KUKA KRL program: Up23.src, Up23.dat

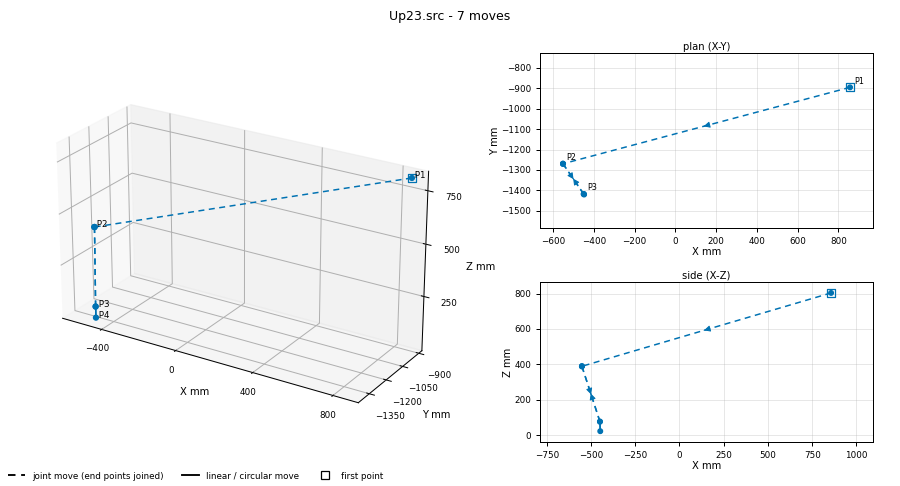
[picture p0: tool path of Up23.src, 7 of 7 moves have a stored position in this frame; points joined in program order, loops and branches not executed]
--- Up23.src ---
&ACCESS RV1
&REL 151
&COMMENT VW380 Ablegen_AFO415600
&PARAM EDITMASK = Up999[1-999]
&PARAM TPVW_VERSION = 8.3.18
&PARAM TEMPLATE = C:\KRC\Roboter\Template\upvorgabe
&PARAM DISKPATH = UPs
DEF UP23()
   ; FOLD UP Anfang;%{SE} %MKUKATPVW
   SPS_N=-1
   SPS_FERTIG=FALSE
   IF NOT CALLBYSELECT THEN
      INTERRUPT DECL 10 WHEN $CYCFLAG[254]==FALSE DO VW(#FB_STOP,TRUE)
      INTERRUPT ON 10
      INT10=TRUE
      VW_USR_R (#USR_INIT)
   ENDIF
   VW(#VW_INIT_UP,TRUE)
   ; ENDFOLD
   ;FOLD -- VW380, THIL -- ;%{PSE}%MKUKATPVW,%CVW_COM,%VCOMMENT,%P 1:Comment:, 2:VW380, THIL
      ;FOLD {H}
         M_COMMENT("VW380, THIL")
      ;ENDFOLD
   ;ENDFOLD
   ;FOLD -- 415600R01 -- ;%{PSE}%MKUKATPVW,%CVW_COM,%VCOMMENT,%P 1:Comment:, 2:415600R01
      ;FOLD {H}
         M_COMMENT("415600R01")
      ;ENDFOLD
   ;ENDFOLD
   ;FOLD -- FRG ST415600 -- ;%{PSE}%MKUKATPVW,%CVW_COM,%VCOMMENT,%P 1:Comment:, 2:FRG ST415600
      ;FOLD {H}
         M_COMMENT("FRG ST415600")
      ;ENDFOLD
   ;ENDFOLD
   ;FOLD -- ACHTUNG! Position ist nicht von PF0 anfahrbar! -- ;%{PSE}%MKUKATPVW,%CVW_COM,%VCOMMENT,%P 1:Comment:, 2:ACHTUNG! Position ist nicht von PF0 anfahrbar!
      ;FOLD {H}
         M_COMMENT("ACHTUNG! Position ist nicht von PF0 anfahrbar!")
      ;ENDFOLD
   ;ENDFOLD
   ;FOLD PTP VB=100% VE=0% ACC=100% RobWzg=11 Base=0 SPSTrig=0[1/100s] P ;%{P}%MKUKATPVW,%CMOVE8,%VPTP,%P 1:1, 2: VB=, 3:100, 4:%, 5: VE=, 6:0, 7:%, 8: ACC=, 9:100, 10:%, 11: RobWzg=, 12:11, 13: Base=, 14:0, 15: SPSTrig=, 16:0, 17:[1/100s], 18: P, 19:1, 20:-1, 21:1
      ;FOLD 1: FB PSPS = EIN ;%{SE}%MKUKATPVW %CVW_SPS %VFBPSPS %P 2:FB PSPS = EIN,3:FBPSPS
      ;ENDFOLD
      ;FOLD 2: A23 = AUS ;%{SE}%MKUKATPVW %CVW_SPS %VBOASG %P 2:A23 = AUS,3:BOASG
      ;ENDFOLD
      ;FOLD 3: t3 ( EIN ) = 0[1/10Sek] ;%{SE}%MKUKATPVW %CVW_SPS %VTASG %P 2:t3 ( EIN ) = 0[1/10Sek],3:TASG
      ;ENDFOLD
      ;FOLD 4: SPSMAKRO50 = EIN ;%{SE}%MKUKATPVW %CVW_SPS %VMAKRO %P 2:SPSMAKRO50 = EIN,3:MAKRO
      ;ENDFOLD
      ;FOLD 5: A43 = AUS ;%{SE}%MKUKATPVW %CVW_SPS %VBOASG %P 2:A43 = AUS,3:BOASG
      ;ENDFOLD
      ;FOLD 6: A44 = AUS ;%{SE}%MKUKATPVW %CVW_SPS %VBOASG %P 2:A44 = AUS,3:BOASG
      ;ENDFOLD
      ;FOLD 7: A65 = AUS ;%{SE}%MKUKATPVW %CVW_SPS %VBOASG %P 2:A65 = AUS,3:BOASG
      ;ENDFOLD
      ;FOLD 8: A68 = EIN ;%{SE}%MKUKATPVW %CVW_SPS %VBOASG %P 2:A68 = EIN,3:BOASG
      ;ENDFOLD
      ;FOLD 9: A69 = AUS ;%{SE}%MKUKATPVW %CVW_SPS %VBOASG %P 2:A69 = AUS,3:BOASG
      ;ENDFOLD
      ;FOLD 10: A71 = AUS ;%{SE}%MKUKATPVW %CVW_SPS %VBOASG %P 2:A71 = AUS,3:BOASG
      ;ENDFOLD
      ;FOLD 11: A72 = EIN ;%{SE}%MKUKATPVW %CVW_SPS %VBOASG %P 2:A72 = EIN,3:BOASG
      ;ENDFOLD
      ;FOLD 12: A73 = AUS ;%{SE}%MKUKATPVW %CVW_SPS %VBOASG %P 2:A73 = AUS,3:BOASG
      ;ENDFOLD
      ;FOLD 13: A76 = EIN ;%{SE}%MKUKATPVW %CVW_SPS %VBOASG %P 2:A76 = EIN,3:BOASG
      ;ENDFOLD
      ;FOLD 14: A77 = AUS ;%{SE}%MKUKATPVW %CVW_SPS %VBOASG %P 2:A77 = AUS,3:BOASG
      ;ENDFOLD
      ;FOLD 15: A80 = EIN ;%{SE}%MKUKATPVW %CVW_SPS %VBOASG %P 2:A80 = EIN,3:BOASG
      ;ENDFOLD
      ;FOLD 16: F930 = AUS ;%{SE}%MKUKATPVW %CVW_SPS %VBOASG %P 2:F930 = AUS,3:BOASG
      ;ENDFOLD
      ;FOLD 17: F939 = AUS ;%{SE}%MKUKATPVW %CVW_SPS %VBOASG %P 2:F939 = AUS,3:BOASG
      ;ENDFOLD
      ;FOLD 18: WARTE BIS E64 & E72 ;%{SE}%MKUKATPVW %CVW_SPS %VWBOASG %P 2:WARTE BIS E64 & E72,3:WBOASG
      ;ENDFOLD
      ;FOLD 19: A72 = AUS ;%{SE}%MKUKATPVW %CVW_SPS %VBOASG %P 2:A72 = AUS,3:BOASG
      ;ENDFOLD
      ;FOLD 20: WARTE BIS E44 & E43 ;%{SE}%MKUKATPVW %CVW_SPS %VWBOASG %P 2:WARTE BIS E44 & E43,3:WBOASG
      ;ENDFOLD
      ;FOLD 21: WARTE BIS E23 ;%{SE}%MKUKATPVW %CVW_SPS %VWBOASG %P 2:WARTE BIS E23,3:WBOASG
      ;ENDFOLD
      ;FOLD 22: A23 = EIN ;%{SE}%MKUKATPVW %CVW_SPS %VBOASG %P 2:A23 = EIN,3:BOASG
      ;ENDFOLD
      ;FOLD 23: FB PSPS = M2 & M30 & M32 & M34 & M63 & M64 & E64 & E72 & E44 & E43 ;%{SE}%MKUKATPVW %CVW_SPS %VFBPSPS %P 2:FB PSPS = M2 & M30 & M32 & M34 & M63 & M64 & E64 & E72 & E44 & E43,3:FBPSPS
      ;ENDFOLD
      ;FOLD {H}
         VW_MPARA_ACT=P1_D
         Act_P1 = P1
         Act_P2 = P1
         VW(#MPARA,TRUE)
         SPS_FERTIG=FALSE
         TRIGGER WHEN DISTANCE=1 DELAY=0 DO SPS_TRIG(1) PRIO=-1
         PTP P1
         $ADVANCE=1
         WAIT FOR SPS_FERTIG
      ;ENDFOLD
   ;ENDFOLD
   ;FOLD PTP VB=100% VE=100% ACC=100% RobWzg=11 Base=0 SPSTrig=0[1/100s] P ;%{P}%MKUKATPVW,%CMOVE8,%VPTP,%P 1:1, 2: VB=, 3:100, 4:%, 5: VE=, 6:100, 7:%, 8: ACC=, 9:100, 10:%, 11: RobWzg=, 12:11, 13: Base=, 14:0, 15: SPSTrig=, 16:0, 17:[1/100s], 18: P, 19:2, 20:-1, 21:2
      ;FOLD 1: FB PSPS = M2 & M30 & M32 & M34 & M63 & M64 & E64 & E72 & E44 & E43 ;%{SE}%MKUKATPVW %CVW_SPS %VFBPSPS %P 2:FB PSPS = M2 & M30 & M32 & M34 & M63 & M64 & E64 & E72 & E44 & E43,3:FBPSPS
      ;ENDFOLD
      ;FOLD {H}
         VW_MPARA_ACT=P2_D
         Act_P1 = P2
         Act_P2 = P2
         VW(#MPARA,TRUE)
         SPS_FERTIG=FALSE
         TRIGGER WHEN DISTANCE=1 DELAY=0 DO SPS_TRIG(10002) PRIO=-1 UP_TIME_OUT=SPS_TIMEOUT
         PTP P2 C_PTP C_VEL
         $ADVANCE=1
      ;ENDFOLD
   ;ENDFOLD
   ;FOLD -- Greifer AUF -- ;%{PSE}%MKUKATPVW,%CVW_COM,%VCOMMENT,%P 1:Comment:, 2:Greifer AUF
      ;FOLD {H}
         M_COMMENT("Greifer AUF")
      ;ENDFOLD
   ;ENDFOLD
   ;FOLD PTP VB=100% VE=0% ACC=100% RobWzg=11 Base=0 SPSTrig=0[1/100s] P ;%{P}%MKUKATPVW,%CMOVE8,%VPTP,%P 1:1, 2: VB=, 3:100, 4:%, 5: VE=, 6:0, 7:%, 8: ACC=, 9:100, 10:%, 11: RobWzg=, 12:11, 13: Base=, 14:0, 15: SPSTrig=, 16:0, 17:[1/100s], 18: P, 19:3, 20:-1, 21:3
      ;FOLD 1: FB PSPS = EIN ;%{SE}%MKUKATPVW %CVW_SPS %VFBPSPS %P 2:FB PSPS = EIN,3:FBPSPS
      ;ENDFOLD
      ;FOLD 2: A23 = AUS ;%{SE}%MKUKATPVW %CVW_SPS %VBOASG %P 2:A23 = AUS,3:BOASG
      ;ENDFOLD
      ;FOLD 3: F1 = EIN ;%{SE}%MKUKATPVW %CVW_SPS %VBOASG %P 2:F1 = EIN,3:BOASG
      ;ENDFOLD
      ;FOLD 4: SPSMAKRO342 = !E15 ;%{SE}%MKUKATPVW %CVW_SPS %VMAKRO %P 2:SPSMAKRO342 = !E15,3:MAKRO
      ;ENDFOLD
      ;FOLD 5: SPSMAKRO340 = EIN ;%{SE}%MKUKATPVW %CVW_SPS %VMAKRO %P 2:SPSMAKRO340 = EIN,3:MAKRO
      ;ENDFOLD
      ;FOLD 6: WARTE BIS E23 & M31 ;%{SE}%MKUKATPVW %CVW_SPS %VWBOASG %P 2:WARTE BIS E23 & M31,3:WBOASG
      ;ENDFOLD
      ;FOLD 7: FB PSPS = M2 & M30 & M31 & M34 & M63 & M64 & E64 & E72 & E44 & E43 ;%{SE}%MKUKATPVW %CVW_SPS %VFBPSPS %P 2:FB PSPS = M2 & M30 & M31 & M34 & M63 & M64 & E64 & E72 & E44 & E43,3:FBPSPS
      ;ENDFOLD
      ;FOLD {H}
         VW_MPARA_ACT=P3_D
         Act_P1 = P3
         Act_P2 = P3
         VW(#MPARA,TRUE)
         SPS_FERTIG=FALSE
         TRIGGER WHEN DISTANCE=1 DELAY=0 DO SPS_TRIG(3) PRIO=-1
         PTP P3
         $ADVANCE=1
         WAIT FOR SPS_FERTIG
      ;ENDFOLD
   ;ENDFOLD
   ;FOLD -- ABL ST415202 -- ;%{PSE}%MKUKATPVW,%CVW_COM,%VCOMMENT,%P 1:Comment:, 2:ABL ST415202
      ;FOLD {H}
         M_COMMENT("ABL ST415202")
      ;ENDFOLD
   ;ENDFOLD
   ;FOLD -- Sauger AUS -- ;%{PSE}%MKUKATPVW,%CVW_COM,%VCOMMENT,%P 1:Comment:, 2:Sauger AUS
      ;FOLD {H}
         M_COMMENT("Sauger AUS")
      ;ENDFOLD
   ;ENDFOLD
   ;FOLD -- FM 2 -- ;%{PSE}%MKUKATPVW,%CVW_COM,%VCOMMENT,%P 1:Comment:, 2:FM 2
      ;FOLD {H}
         M_COMMENT("FM 2")
      ;ENDFOLD
   ;ENDFOLD
   ;FOLD LIN VB=250[mm/s] VE=0% ACC=100% RobWzg=11 Base=0 SPSTrig=5[1/100s] P ;%{P}%MKUKATPVW,%CMOVE8,%VLIN,%P 1:2, 2: VB=, 3:250, 4:[mm/s], 5: VE=, 6:0, 7:%, 8: ACC=, 9:100, 10:%, 11: RobWzg=, 12:11, 13: Base=, 14:0, 15: SPSTrig=, 16:5, 17:[1/100s], 18: P, 19:4, 20:-1, 21:4
      ;FOLD 1: FB PSPS = EIN ;%{SE}%MKUKATPVW %CVW_SPS %VFBPSPS %P 2:FB PSPS = EIN,3:FBPSPS
      ;ENDFOLD
      ;FOLD 2: A23 = AUS ;%{SE}%MKUKATPVW %CVW_SPS %VBOASG %P 2:A23 = AUS,3:BOASG
      ;ENDFOLD
      ;FOLD 3: A69 = EIN ;%{SE}%MKUKATPVW %CVW_SPS %VBOASG %P 2:A69 = EIN,3:BOASG
      ;ENDFOLD
      ;FOLD 4: A71 = EIN ;%{SE}%MKUKATPVW %CVW_SPS %VBOASG %P 2:A71 = EIN,3:BOASG
      ;ENDFOLD
      ;FOLD 5: F17 = !E15 ;%{SE}%MKUKATPVW %CVW_SPS %VBOASG %P 2:F17 = !E15,3:BOASG
      ;ENDFOLD
      ;FOLD 6: F18 = !E15 ;%{SE}%MKUKATPVW %CVW_SPS %VBOASG %P 2:F18 = !E15,3:BOASG
      ;ENDFOLD
      ;FOLD 7: SPSMAKRO342 = !E15 ;%{SE}%MKUKATPVW %CVW_SPS %VMAKRO %P 2:SPSMAKRO342 = !E15,3:MAKRO
      ;ENDFOLD
      ;FOLD 8: SPSMAKRO340 = EIN ;%{SE}%MKUKATPVW %CVW_SPS %VMAKRO %P 2:SPSMAKRO340 = EIN,3:MAKRO
      ;ENDFOLD
      ;FOLD 9: SPSMAKRO2 = EIN ;%{SE}%MKUKATPVW %CVW_SPS %VMAKRO %P 2:SPSMAKRO2 = EIN,3:MAKRO
      ;ENDFOLD
      ;FOLD 10: WARTE BIS M13 & M31 & E63 & E72 ;%{SE}%MKUKATPVW %CVW_SPS %VWBOASG %P 2:WARTE BIS M13 & M31 & E63 & E72,3:WBOASG
      ;ENDFOLD
      ;FOLD 11: A69 = AUS ;%{SE}%MKUKATPVW %CVW_SPS %VBOASG %P 2:A69 = AUS,3:BOASG
      ;ENDFOLD
      ;FOLD 12: A71 = AUS ;%{SE}%MKUKATPVW %CVW_SPS %VBOASG %P 2:A71 = AUS,3:BOASG
      ;ENDFOLD
      ;FOLD 13: WARTE BIS E23 ;%{SE}%MKUKATPVW %CVW_SPS %VWBOASG %P 2:WARTE BIS E23,3:WBOASG
      ;ENDFOLD
      ;FOLD 14: A23 = EIN ;%{SE}%MKUKATPVW %CVW_SPS %VBOASG %P 2:A23 = EIN,3:BOASG
      ;ENDFOLD
      ;FOLD 15: FB PSPS = M13 & M30 & M31 & M34 & E63 & E72 & E44 & E43 ;%{SE}%MKUKATPVW %CVW_SPS %VFBPSPS %P 2:FB PSPS = M13 & M30 & M31 & M34 & E63 & E72 & E44 & E43,3:FBPSPS
      ;ENDFOLD
      ;FOLD {H}
         VW_MPARA_ACT=P4_D
         Act_P1 = P4
         Act_P2 = P4
         VW(#MPARA,TRUE)
         SPS_FERTIG=FALSE
         TRIGGER WHEN DISTANCE=1 DELAY=-50 DO SPS_TRIG(4) PRIO=-1
         LIN P4
         $ADVANCE=1
         WAIT FOR SPS_FERTIG
      ;ENDFOLD
   ;ENDFOLD
   ;FOLD -- PF ST415600 -- ;%{PSE}%MKUKATPVW,%CVW_COM,%VCOMMENT,%P 1:Comment:, 2:PF ST415600
      ;FOLD {H}
         M_COMMENT("PF ST415600")
      ;ENDFOLD
   ;ENDFOLD
   ;FOLD LIN VB=250[mm/s] VE=100% ACC=100% RobWzg=11 Base=0 SPSTrig=0[1/100s] P ;%{P}%MKUKATPVW,%CMOVE8,%VLIN,%P 1:2, 2: VB=, 3:250, 4:[mm/s], 5: VE=, 6:100, 7:%, 8: ACC=, 9:100, 10:%, 11: RobWzg=, 12:11, 13: Base=, 14:0, 15: SPSTrig=, 16:0, 17:[1/100s], 18: P, 19:5, 20:-1, 21:5
      ;FOLD 1: FB PSPS = EIN ;%{SE}%MKUKATPVW %CVW_SPS %VFBPSPS %P 2:FB PSPS = EIN,3:FBPSPS
      ;ENDFOLD
      ;FOLD 2: A72 = EIN ;%{SE}%MKUKATPVW %CVW_SPS %VBOASG %P 2:A72 = EIN,3:BOASG
      ;ENDFOLD
      ;FOLD 3: A577 = EIN ;%{SE}%MKUKATPVW %CVW_SPS %VBOASG %P 2:A577 = EIN,3:BOASG
      ;ENDFOLD
      ;FOLD 4: Puls A579 = Pegel:EIN Zeit:10 [1/10Sek] ;%{SE}%MKUKATPVW %CVW_SPS %VPULS %P 2:Puls A579 = Pegel:EIN Zeit:10 [1/10Sek],3:PULS
      ;ENDFOLD
      ;FOLD 5: FB PSPS = M13 & M30 & M34 & E44 & E43 ;%{SE}%MKUKATPVW %CVW_SPS %VFBPSPS %P 2:FB PSPS = M13 & M30 & M34 & E44 & E43,3:FBPSPS
      ;ENDFOLD
      ;FOLD {H}
         VW_MPARA_ACT=P5_D
         Act_P1 = P5
         Act_P2 = P5
         VW(#MPARA,TRUE)
         SPS_FERTIG=FALSE
         TRIGGER WHEN DISTANCE=1 DELAY=0 DO SPS_TRIG(10005) PRIO=-1 UP_TIME_OUT=SPS_TIMEOUT
         LIN P5 C_VEL
         $ADVANCE=1
      ;ENDFOLD
   ;ENDFOLD
   ;FOLD PTP VB=100% VE=100% ACC=100% RobWzg=11 Base=0 SPSTrig=0[1/100s] P ;%{P}%MKUKATPVW,%CMOVE8,%VPTP,%P 1:1, 2: VB=, 3:100, 4:%, 5: VE=, 6:100, 7:%, 8: ACC=, 9:100, 10:%, 11: RobWzg=, 12:11, 13: Base=, 14:0, 15: SPSTrig=, 16:0, 17:[1/100s], 18: P, 19:6, 20:-1, 21:6
      ;FOLD 1: FB PSPS = M13 & M30 & M34 & E44 & E43 ;%{SE}%MKUKATPVW %CVW_SPS %VFBPSPS %P 2:FB PSPS = M13 & M30 & M34 & E44 & E43,3:FBPSPS
      ;ENDFOLD
      ;FOLD {H}
         VW_MPARA_ACT=P6_D
         Act_P1 = P6
         Act_P2 = P6
         VW(#MPARA,TRUE)
         SPS_FERTIG=FALSE
         TRIGGER WHEN DISTANCE=1 DELAY=0 DO SPS_TRIG(10006) PRIO=-1 UP_TIME_OUT=SPS_TIMEOUT
         PTP P6 C_PTP C_VEL
         $ADVANCE=1
      ;ENDFOLD
   ;ENDFOLD
   ;FOLD PTP VB=100% VE=0% ACC=100% RobWzg=11 Base=0 SPSTrig=0[1/100s] P ;%{P}%MKUKATPVW,%CMOVE8,%VPTP,%P 1:1, 2: VB=, 3:100, 4:%, 5: VE=, 6:0, 7:%, 8: ACC=, 9:100, 10:%, 11: RobWzg=, 12:11, 13: Base=, 14:0, 15: SPSTrig=, 16:0, 17:[1/100s], 18: P, 19:7, 20:-1, 21:7
      ;FOLD 1: FB PSPS = EIN ;%{SE}%MKUKATPVW %CVW_SPS %VFBPSPS %P 2:FB PSPS = EIN,3:FBPSPS
      ;ENDFOLD
      ;FOLD 2: A23 = AUS ;%{SE}%MKUKATPVW %CVW_SPS %VBOASG %P 2:A23 = AUS,3:BOASG
      ;ENDFOLD
      ;FOLD 3: t3 ( EIN) = STOP ;%{SE}%MKUKATPVW %CVW_SPS %VTSTOP %P 2:t3 ( EIN) = STOP,3:TSTOP
      ;ENDFOLD
      ;FOLD 4: WARTE BIS E23 ;%{SE}%MKUKATPVW %CVW_SPS %VWBOASG %P 2:WARTE BIS E23,3:WBOASG
      ;ENDFOLD
      ;FOLD 5: A23 = EIN ;%{SE}%MKUKATPVW %CVW_SPS %VBOASG %P 2:A23 = EIN,3:BOASG
      ;ENDFOLD
      ;FOLD 6: FB PSPS = M13 & M30 & M34 & E43 & E44 ;%{SE}%MKUKATPVW %CVW_SPS %VFBPSPS %P 2:FB PSPS = M13 & M30 & M34 & E43 & E44,3:FBPSPS
      ;ENDFOLD
      ;FOLD {H}
         VW_MPARA_ACT=P7_D
         Act_P1 = P7
         Act_P2 = P7
         VW(#MPARA,TRUE)
         SPS_FERTIG=FALSE
         TRIGGER WHEN DISTANCE=1 DELAY=0 DO SPS_TRIG(7) PRIO=-1
         PTP P7
         $ADVANCE=1
         WAIT FOR SPS_FERTIG
      ;ENDFOLD
   ;ENDFOLD
   ; FOLD ;%{H}
END
DEF SPS_TRIG(NO :IN)
   INT NO
   INT VW_STOP
   BOOL UES
   BOOL ANA_UES
   BOOL ANA_TRIG
   VW_STOP=$VW_PSPS_STOP
   UES=FALSE
   ANA_UES=FALSE
   ANA_TRIG=FALSE
   IF ((NO>10000) AND (NO<20000)) THEN
      NO=NO-10000
      UES=TRUE
   ENDIF
   IF ((NO>20000) AND (NO<30000)) THEN
      NO=NO-20000
      ANA_TRIG=TRUE
   ENDIF
   IF NO>30000 THEN
      NO=NO-30000
      ANA_UES=TRUE
      ANA_TRIG=TRUE
   ENDIF
   ; FOLD ;%{H}
   IF ((VW_STOP B_AND 'B0001') > 0) THEN
      ;-- Trigger vorzeitig geschaltet (delay < 0) oder MStep
      IF (((VW_STOP B_AND 'B0110') > 0) AND ($MODE_OP<>#EX)) THEN
         ;-- MStep oder BCO Bewegung
         HALT
      ENDIF
   ENDIF
   ; ENDFOLD
   IF (SEARCH_END) THEN
      SEARCH_END = FALSE
      INTERRUPT OFF 39
   ENDIF
   SWITCH NO
      CASE 1
         ;FOLD SPS_TRIG1 {H}
            VALCYCFL30=$CYCFLAG[254]
            $CYCFLAG[254]=(TRUE) AND $CYCFLAG[255] OR ($TIMER[61]<0)
            VW(#FB_CHECK,TRUE)
            $OUT[23] = FALSE
            VW(#SET_TIME,TRUE,3,0,0)
            SEL_RES=SELECT(#MAKRO,50,TRUE,,,,,FALSE)
            $OUT[43] = FALSE
            $OUT[44] = FALSE
            $OUT[65] = FALSE
            $OUT[68] = TRUE
            $OUT[69] = FALSE
            $OUT[71] = FALSE
            $OUT[72] = TRUE
            $OUT[73] = FALSE
            $OUT[76] = TRUE
            $OUT[77] = FALSE
            $OUT[80] = TRUE
            $FLAG[930] = FALSE
            $FLAG[939] = FALSE
            $LOOP_MSG[]="E64 & E72"
            $LOOP_CONT=TRUE
            WAIT FOR ($IN[64] AND $IN[72]) OR (NOT $LOOP_CONT AND ($MODE_OP<>#EX))
            $LOOP_MSG[]="                                                                                                                                "
            $OUT[72] = FALSE
            $LOOP_MSG[]="E44 & E43"
            $LOOP_CONT=TRUE
            WAIT FOR ($IN[44] AND $IN[43]) OR (NOT $LOOP_CONT AND ($MODE_OP<>#EX))
            $LOOP_MSG[]="                                                                                                                                "
            $LOOP_MSG[]="E23"
            $LOOP_CONT=TRUE
            WAIT FOR ($IN[23]) OR (NOT $LOOP_CONT AND ($MODE_OP<>#EX))
            $LOOP_MSG[]="                                                                                                                                "
            $OUT[23] = TRUE
            VALCYCFL30=$CYCFLAG[254]
            $CYCFLAG[254]=($CYCFLAG[2] AND $CYCFLAG[30] AND $CYCFLAG[32] AND $CYCFLAG[34] AND $CYCFLAG[63] AND $CYCFLAG[64] AND $IN[64] AND $IN[72] AND $IN[44] AND $IN[43]) AND $CYCFLAG[255] OR ($TIMER[61]<0)
            VW(#FB_CHECK,TRUE)
         ;ENDFOLD
      CASE 2
         ;FOLD SPS_TRIG2 {H}
            VALCYCFL30=$CYCFLAG[254]
            $CYCFLAG[254]=($CYCFLAG[2] AND $CYCFLAG[30] AND $CYCFLAG[32] AND $CYCFLAG[34] AND $CYCFLAG[63] AND $CYCFLAG[64] AND $IN[64] AND $IN[72] AND $IN[44] AND $IN[43]) AND $CYCFLAG[255] OR ($TIMER[61]<0)
            VW(#FB_CHECK,TRUE)
         ;ENDFOLD
      CASE 3
         ;FOLD SPS_TRIG3 {H}
            VALCYCFL30=$CYCFLAG[254]
            $CYCFLAG[254]=(TRUE) AND $CYCFLAG[255] OR ($TIMER[61]<0)
            VW(#FB_CHECK,TRUE)
            $OUT[23] = FALSE
            $FLAG[1] = TRUE
            SEL_RES=SELECT(#MAKRO,342,NOT $IN[15],,,,,FALSE)
            SEL_RES=SELECT(#MAKRO,340,TRUE,,,,,FALSE)
            $LOOP_MSG[]="E23 & M31"
            $LOOP_CONT=TRUE
            WAIT FOR ($IN[23] AND $CYCFLAG[31]) OR (NOT $LOOP_CONT AND ($MODE_OP<>#EX))
            $LOOP_MSG[]="                                                                                                                                "
            VALCYCFL30=$CYCFLAG[254]
            $CYCFLAG[254]=($CYCFLAG[2] AND $CYCFLAG[30] AND $CYCFLAG[31] AND $CYCFLAG[34] AND $CYCFLAG[63] AND $CYCFLAG[64] AND $IN[64] AND $IN[72] AND $IN[44] AND $IN[43]) AND $CYCFLAG[255] OR ($TIMER[61]<0)
            VW(#FB_CHECK,TRUE)
         ;ENDFOLD
      CASE 4
         ;FOLD SPS_TRIG4 {H}
            VALCYCFL30=$CYCFLAG[254]
            $CYCFLAG[254]=(TRUE) AND $CYCFLAG[255] OR ($TIMER[61]<0)
            VW(#FB_CHECK,TRUE)
            $OUT[23] = FALSE
            $OUT[69] = TRUE
            $OUT[71] = TRUE
            $FLAG[17] = NOT $IN[15]
            $FLAG[18] = NOT $IN[15]
            SEL_RES=SELECT(#MAKRO,342,NOT $IN[15],,,,,FALSE)
            SEL_RES=SELECT(#MAKRO,340,TRUE,,,,,FALSE)
            SEL_RES=SELECT(#MAKRO,2,TRUE,,,,,FALSE)
            $LOOP_MSG[]="M13 & M31 & E63 & E72"
            $LOOP_CONT=TRUE
            WAIT FOR ($CYCFLAG[13] AND $CYCFLAG[31] AND $IN[63] AND $IN[72]) OR (NOT $LOOP_CONT AND ($MODE_OP<>#EX))
            $LOOP_MSG[]="                                                                                                                                "
            $OUT[69] = FALSE
            $OUT[71] = FALSE
            $LOOP_MSG[]="E23"
            $LOOP_CONT=TRUE
            WAIT FOR ($IN[23]) OR (NOT $LOOP_CONT AND ($MODE_OP<>#EX))
            $LOOP_MSG[]="                                                                                                                                "
            $OUT[23] = TRUE
            VALCYCFL30=$CYCFLAG[254]
            $CYCFLAG[254]=($CYCFLAG[13] AND $CYCFLAG[30] AND $CYCFLAG[31] AND $CYCFLAG[34] AND $IN[63] AND $IN[72] AND $IN[44] AND $IN[43]) AND $CYCFLAG[255] OR ($TIMER[61]<0)
            VW(#FB_CHECK,TRUE)
         ;ENDFOLD
      CASE 5
         ;FOLD SPS_TRIG5 {H}
            VALCYCFL30=$CYCFLAG[254]
            $CYCFLAG[254]=(TRUE) AND $CYCFLAG[255] OR ($TIMER[61]<0)
            VW(#FB_CHECK,TRUE)
            $OUT[72] = TRUE
            $OUT[577] = TRUE
            VW(#VW_PULSE, TRUE, 1, 0, 10, 579, TRUE)
            VALCYCFL30=$CYCFLAG[254]
            $CYCFLAG[254]=($CYCFLAG[13] AND $CYCFLAG[30] AND $CYCFLAG[34] AND $IN[44] AND $IN[43]) AND $CYCFLAG[255] OR ($TIMER[61]<0)
            VW(#FB_CHECK,TRUE)
         ;ENDFOLD
      CASE 6
         ;FOLD SPS_TRIG6 {H}
            VALCYCFL30=$CYCFLAG[254]
            $CYCFLAG[254]=($CYCFLAG[13] AND $CYCFLAG[30] AND $CYCFLAG[34] AND $IN[44] AND $IN[43]) AND $CYCFLAG[255] OR ($TIMER[61]<0)
            VW(#FB_CHECK,TRUE)
         ;ENDFOLD
      CASE 7
         ;FOLD SPS_TRIG7 {H}
            VALCYCFL30=$CYCFLAG[254]
            $CYCFLAG[254]=(TRUE) AND $CYCFLAG[255] OR ($TIMER[61]<0)
            VW(#FB_CHECK,TRUE)
            $OUT[23] = FALSE
            VW(#SET_TIME,TRUE,3,1,0)
            $LOOP_MSG[]="E23"
            $LOOP_CONT=TRUE
            WAIT FOR ($IN[23]) OR (NOT $LOOP_CONT AND ($MODE_OP<>#EX))
            $LOOP_MSG[]="                                                                                                                                "
            $OUT[23] = TRUE
            VALCYCFL30=$CYCFLAG[254]
            $CYCFLAG[254]=($CYCFLAG[13] AND $CYCFLAG[30] AND $CYCFLAG[34] AND $IN[43] AND $IN[44]) AND $CYCFLAG[255] OR ($TIMER[61]<0)
            VW(#FB_CHECK,TRUE)
         ;ENDFOLD
      CASE 8
         ;FOLD SPS_TRIG8 {H}
         ;ENDFOLD
      CASE 9
         ;FOLD SPS_TRIG9 {H}
         ;ENDFOLD
      CASE 10
         ;FOLD SPS_TRIG10 {H}
         ;ENDFOLD
      CASE 11
         ;FOLD SPS_TRIG11 {H}
         ;ENDFOLD
      CASE 12
         ;FOLD SPS_TRIG12 {H}
         ;ENDFOLD
      CASE 13
         ;FOLD SPS_TRIG13 {H}
         ;ENDFOLD
      CASE 14
         ;FOLD SPS_TRIG14 {H}
         ;ENDFOLD
      CASE 15
         ;FOLD SPS_TRIG15 {H}
         ;ENDFOLD
      CASE 16
         ;FOLD SPS_TRIG16 {H}
         ;ENDFOLD
      CASE 17
         ;FOLD SPS_TRIG17 {H}
         ;ENDFOLD
      CASE 18
         ;FOLD SPS_TRIG18 {H}
         ;ENDFOLD
      CASE 19
         ;FOLD SPS_TRIG19 {H}
         ;ENDFOLD
      CASE 20
         ;FOLD SPS_TRIG20 {H}
         ;ENDFOLD
      CASE 21
         ;FOLD SPS_TRIG21 {H}
         ;ENDFOLD
      CASE 22
         ;FOLD SPS_TRIG22 {H}
         ;ENDFOLD
      CASE 23
         ;FOLD SPS_TRIG23 {H}
         ;ENDFOLD
      CASE 24
         ;FOLD SPS_TRIG24 {H}
         ;ENDFOLD
      CASE 25
         ;FOLD SPS_TRIG25 {H}
         ;ENDFOLD
      CASE 26
         ;FOLD SPS_TRIG26 {H}
         ;ENDFOLD
      CASE 27
         ;FOLD SPS_TRIG27 {H}
         ;ENDFOLD
      CASE 28
         ;FOLD SPS_TRIG28 {H}
         ;ENDFOLD
      CASE 29
         ;FOLD SPS_TRIG29 {H}
         ;ENDFOLD
      CASE 30
         ;FOLD SPS_TRIG30 {H}
         ;ENDFOLD
      CASE 31
         ;FOLD SPS_TRIG31 {H}
         ;ENDFOLD
      CASE 32
         ;FOLD SPS_TRIG32 {H}
         ;ENDFOLD
      CASE 33
         ;FOLD SPS_TRIG33 {H}
         ;ENDFOLD
      CASE 34
         ;FOLD SPS_TRIG34 {H}
         ;ENDFOLD
      CASE 35
         ;FOLD SPS_TRIG35 {H}
         ;ENDFOLD
      CASE 36
         ;FOLD SPS_TRIG36 {H}
         ;ENDFOLD
      CASE 37
         ;FOLD SPS_TRIG37 {H}
         ;ENDFOLD
      CASE 38
         ;FOLD SPS_TRIG38 {H}
         ;ENDFOLD
      CASE 39
         ;FOLD SPS_TRIG39 {H}
         ;ENDFOLD
      CASE 40
         ;FOLD SPS_TRIG40 {H}
         ;ENDFOLD
      CASE 41
         ;FOLD SPS_TRIG41 {H}
         ;ENDFOLD
      CASE 42
         ;FOLD SPS_TRIG42 {H}
         ;ENDFOLD
      CASE 43
         ;FOLD SPS_TRIG43 {H}
         ;ENDFOLD
      CASE 44
         ;FOLD SPS_TRIG44 {H}
         ;ENDFOLD
      CASE 45
         ;FOLD SPS_TRIG45 {H}
         ;ENDFOLD
      CASE 46
         ;FOLD SPS_TRIG46 {H}
         ;ENDFOLD
      CASE 47
         ;FOLD SPS_TRIG47 {H}
         ;ENDFOLD
      CASE 48
         ;FOLD SPS_TRIG48 {H}
         ;ENDFOLD
      CASE 49
         ;FOLD SPS_TRIG49 {H}
         ;ENDFOLD
      CASE 50
         ;FOLD SPS_TRIG50 {H}
         ;ENDFOLD
      CASE 51
         ;FOLD SPS_TRIG51 {H}
         ;ENDFOLD
      CASE 52
         ;FOLD SPS_TRIG52 {H}
         ;ENDFOLD
      CASE 53
         ;FOLD SPS_TRIG53 {H}
         ;ENDFOLD
      CASE 54
         ;FOLD SPS_TRIG54 {H}
         ;ENDFOLD
      CASE 55
         ;FOLD SPS_TRIG55 {H}
         ;ENDFOLD
      CASE 56
         ;FOLD SPS_TRIG56 {H}
         ;ENDFOLD
      CASE 57
         ;FOLD SPS_TRIG57 {H}
         ;ENDFOLD
      CASE 58
         ;FOLD SPS_TRIG58 {H}
         ;ENDFOLD
      CASE 59
         ;FOLD SPS_TRIG59 {H}
         ;ENDFOLD
      CASE 60
         ;FOLD SPS_TRIG60 {H}
         ;ENDFOLD
      CASE 61
         ;FOLD SPS_TRIG61 {H}
         ;ENDFOLD
      CASE 62
         ;FOLD SPS_TRIG62 {H}
         ;ENDFOLD
      CASE 63
         ;FOLD SPS_TRIG63 {H}
         ;ENDFOLD
      CASE 64
         ;FOLD SPS_TRIG64 {H}
         ;ENDFOLD
      CASE 65
         ;FOLD SPS_TRIG65 {H}
         ;ENDFOLD
      CASE 66
         ;FOLD SPS_TRIG66 {H}
         ;ENDFOLD
      CASE 67
         ;FOLD SPS_TRIG67 {H}
         ;ENDFOLD
      CASE 68
         ;FOLD SPS_TRIG68 {H}
         ;ENDFOLD
      CASE 69
         ;FOLD SPS_TRIG69 {H}
         ;ENDFOLD
      CASE 70
         ;FOLD SPS_TRIG70 {H}
         ;ENDFOLD
      CASE 71
         ;FOLD SPS_TRIG71 {H}
         ;ENDFOLD
      CASE 72
         ;FOLD SPS_TRIG72 {H}
         ;ENDFOLD
      CASE 73
         ;FOLD SPS_TRIG73 {H}
         ;ENDFOLD
      CASE 74
         ;FOLD SPS_TRIG74 {H}
         ;ENDFOLD
      CASE 75
         ;FOLD SPS_TRIG75 {H}
         ;ENDFOLD
      CASE 76
         ;FOLD SPS_TRIG76 {H}
         ;ENDFOLD
      CASE 77
         ;FOLD SPS_TRIG77 {H}
         ;ENDFOLD
      CASE 78
         ;FOLD SPS_TRIG78 {H}
         ;ENDFOLD
      CASE 79
         ;FOLD SPS_TRIG79 {H}
         ;ENDFOLD
      CASE 80
         ;FOLD SPS_TRIG80 {H}
         ;ENDFOLD
      CASE 81
         ;FOLD SPS_TRIG81 {H}
         ;ENDFOLD
      CASE 82
         ;FOLD SPS_TRIG82 {H}
         ;ENDFOLD
      CASE 83
         ;FOLD SPS_TRIG83 {H}
         ;ENDFOLD
      CASE 84
         ;FOLD SPS_TRIG84 {H}
         ;ENDFOLD
      CASE 85
         ;FOLD SPS_TRIG85 {H}
         ;ENDFOLD
      CASE 86
         ;FOLD SPS_TRIG86 {H}
         ;ENDFOLD
      CASE 87
         ;FOLD SPS_TRIG87 {H}
         ;ENDFOLD
      CASE 88
         ;FOLD SPS_TRIG88 {H}
         ;ENDFOLD
      CASE 89
         ;FOLD SPS_TRIG89 {H}
         ;ENDFOLD
      CASE 90
         ;FOLD SPS_TRIG90 {H}
         ;ENDFOLD
      CASE 91
         ;FOLD SPS_TRIG91 {H}
         ;ENDFOLD
      CASE 92
         ;FOLD SPS_TRIG92 {H}
         ;ENDFOLD
      CASE 93
         ;FOLD SPS_TRIG93 {H}
         ;ENDFOLD
      CASE 94
         ;FOLD SPS_TRIG94 {H}
         ;ENDFOLD
      CASE 95
         ;FOLD SPS_TRIG95 {H}
         ;ENDFOLD
      CASE 96
         ;FOLD SPS_TRIG96 {H}
         ;ENDFOLD
      CASE 97
         ;FOLD SPS_TRIG97 {H}
         ;ENDFOLD
      CASE 98
         ;FOLD SPS_TRIG98 {H}
         ;ENDFOLD
      CASE 99
         ;FOLD SPS_TRIG99 {H}
         ;ENDFOLD
      CASE 100
         ;FOLD SPS_TRIG100 {H}
         ;ENDFOLD
      CASE 101
         ;FOLD SPS_TRIG101 {H}
         ;ENDFOLD
      CASE 102
         ;FOLD SPS_TRIG102 {H}
         ;ENDFOLD
      CASE 103
         ;FOLD SPS_TRIG103 {H}
         ;ENDFOLD
      CASE 104
         ;FOLD SPS_TRIG104 {H}
         ;ENDFOLD
      CASE 105
         ;FOLD SPS_TRIG105 {H}
         ;ENDFOLD
      CASE 106
         ;FOLD SPS_TRIG106 {H}
         ;ENDFOLD
      CASE 107
         ;FOLD SPS_TRIG107 {H}
         ;ENDFOLD
      CASE 108
         ;FOLD SPS_TRIG108 {H}
         ;ENDFOLD
   DEFAULT
   ENDSWITCH
   ; FOLD ;%{H}
   IF ($MODE_OP<>#EX) THEN
      ;-- Trigger erst nach Wiederanstart geschaltet --
      IF ((((VW_STOP B_AND 'B10010') >0) AND ((VW_STOP B_AND 'B0001')<=0))) THEN
         ;-- MStep Bewegung --
         HALT
      ENDIF
   ENDIF
   ; ENDFOLD
   IF (NOT UES AND NOT ANA_TRIG) THEN
      SPS_FERTIG=TRUE
   ENDIF
   IF (NOT ANA_UES AND ANA_TRIG) THEN
      SPS_FERTIG_ANA=TRUE
   ENDIF
END
; ENDFOLD

--- Up23.dat ---
&ACCESS RV1
&REL 151
&COMMENT VW380 Ablegen_AFO415600
&PARAM EDITMASK = Up999[1-999]
&PARAM TPVW_VERSION = 8.3.18
&PARAM TEMPLATE = C:\KRC\Roboter\Template\upvorgabe
&PARAM DISKPATH = UPs
DEFDAT  Up23
; FOLD ;%{H} %MKUKATPVW
; ENDFOLD
; interface to basic routines
EXT  BAS (BAS_COMMAND  :IN,REAL  :IN )
; interface to VW-standard routines
EXT  VW (VW_COMMAND  :IN,BOOL  :IN,REAL  :IN,REAL  :IN,REAL  :IN,REAL  :IN,BOOL  :IN,E6POS  :IN )
; interface to VW_USER - Call
EXT  VW_USER (VW_USER_CMD  :IN,INT  :IN,REAL  :IN,REAL  :IN,REAL  :IN,REAL  :IN,REAL  :IN,REAL  :IN,REAL  :IN,REAL  :IN,REAL  :IN,BOOL  :IN )
EXT  VW_USR_R (VW_USER_CMD  :IN,INT  :IN,REAL  :IN,REAL  :IN,REAL  :IN,REAL  :IN,REAL  :IN,REAL  :IN,REAL  :IN,REAL  :IN,REAL  :IN,BOOL  :IN )
EXT  IBGN (IBGN_COMMAND  :IN,BOOL  :IN,REAL  :IN,REAL  :IN,BOOL  :IN,E6POS  :OUT )
; interface select routine
EXTFCT  INT  SELECT(SUBTYPE  :IN,INT  :IN,BOOL  :IN,ARI_TYP  :IN,INT  :IN,BOOL_TYP  :IN,INT  :IN,BOOL  :IN)
INT VW_NEXT_FREE=8
INT VW_NFREE_SPS=8
INT VW_MAX_SPS=108
DECL VW_MPARA_TYP P1_D={TOOL_NO 11,BASE_NO 0,VB 100,VE 0,ACC 100,TRG_TIME 0,MOVE_TYPE #PTP_MOTION}
DECL E6POS P1={X 856.774170,Y -895.088684,Z 803.217712,A 3.27273607,B 3.01466203,C 179.931107,S 2,T 2,E1 0.0,E2 0.0,E3 0.0,E4 0.0,E5 0.0,E6 0.0}
DECL VW_MPARA_TYP P2_D={TOOL_NO 11,BASE_NO 0,VB 100,VE 100,ACC 100,TRG_TIME 0,MOVE_TYPE #PTP_MOTION}
DECL E6POS P2={X -551.241882,Y -1269.86902,Z 388.743713,A -51.5507088,B 56.2558517,C 135.690506,S 2,T 2,E1 0.0,E2 0.0,E3 0.0,E4 0.0,E5 0.0,E6 0.0}
DECL VW_MPARA_TYP P3_D={TOOL_NO 11,BASE_NO 0,VB 100,VE 0,ACC 100,TRG_TIME 0,MOVE_TYPE #PTP_MOTION}
DECL E6POS P3={X -449.427185,Y -1418.46204,Z 76.0931702,A -128.567795,B 88.0757294,C 50.9166298,S 2,T 2,E1 0.0,E2 0.0,E3 0.0,E4 0.0,E5 0.0,E6 0.0}
DECL VW_MPARA_TYP P4_D={TOOL_NO 11,BASE_NO 0,VB 250,VE 0,ACC 100,TRG_TIME 5,MOVE_TYPE #PATH_MOTION}
DECL E6POS P4={X -447.588501,Y -1420.88696,Z 21.9472103,A -118.219398,B 87.4826202,C 61.7327919,S 2,T 2,E1 0.0,E2 0.0,E3 0.0,E4 0.0,E5 0.0,E6 0.0}
DECL VW_MPARA_TYP P5_D={TOOL_NO 11,BASE_NO 0,VB 250,VE 100,ACC 100,TRG_TIME 0,MOVE_TYPE #PATH_MOTION}
DECL E6POS P5={X -449.427185,Y -1418.46204,Z 76.0931702,A -128.567795,B 88.0757294,C 50.9166298,S 2,T 2,E1 0.0,E2 0.0,E3 0.0,E4 0.0,E5 0.0,E6 0.0}
DECL VW_MPARA_TYP P6_D={TOOL_NO 11,BASE_NO 0,VB 100,VE 100,ACC 100,TRG_TIME 0,MOVE_TYPE #PTP_MOTION}
DECL E6POS P6={X -551.241882,Y -1269.86902,Z 388.743713,A -51.5507088,B 56.2558517,C 135.690506,S 2,T 2,E1 0.0,E2 0.0,E3 0.0,E4 0.0,E5 0.0,E6 0.0}
DECL VW_MPARA_TYP P7_D={TOOL_NO 11,BASE_NO 0,VB 100,VE 0,ACC 100,TRG_TIME 0,MOVE_TYPE #PTP_MOTION}
DECL E6POS P7={X -551.241882,Y -1269.86902,Z 388.743713,A -51.5507088,B 56.2558517,C 135.690506,S 2,T 2,E1 0.0,E2 0.0,E3 0.0,E4 0.0,E5 0.0,E6 0.0}
ENDDAT
